TYPE typeStationComplexityBuffer :
STRUCT
	buffer: ARRAY[0..2048] OF BYTE;
	
	
END_STRUCT
END_TYPE

(* stored: Version 1.1.0.1, ProductVersion 3.1.4024.12
   DUT typeStationComplexityBuffer: Id {08ccc68b-86a9-4dd5-8617-6cd4fea55199} *)
